FUNCTION_BLOCK StateObserver
VAR_INPUT
	xRobotPoseCam : RobotPose :=[-1, -1, -1];
	xRobotVelocities : RobotVelocities := [0, 0, 0];
END_VAR
VAR_OUTPUT
	yRobotPose : RobotPose;
END_VAR
VAR
END_VAR

END_FUNCTION_BLOCK

(* stored: Version 1.1.0.1, ProductVersion 3.1.4024.11
   POU StateObserver: Id {039231fe-9cf2-4974-9a44-025359184cf4}, SpecialFunc None *)
